FUNCTION_BLOCK FB_Dog EXTENDS FB_Animal
VAR
 
END_VAR

METHOD M_Eat : BOOL
VAR_INPUT
END_VAR
THIS^.sOutput := 'Dog eats dog food';
END_METHOD

END_FUNCTION_BLOCK

(* stored: Version 1.1.0.1, ProductVersion 3.1.4024.16
   POU FB_Dog: Id {fd0858ef-98bf-4118-9af0-63968e61b15b}, SpecialFunc None
   Method M_Eat: Id {c06eeb9a-8a57-4d8b-98f8-93e243548849} *)
